{attribute 'linkalways'} 
{attribute 'no_explicit_call' := 'This FB is a CLASS and must be accessed using methods or properties'}
{attribute 'enable_dynamic_creation'}
FUNCTION_BLOCK Node_ContainerType_Vector_ITcVnImage EXTENDS Node
VAR
    out : _GUID;
END_VAR

METHOD PUBLIC  Clone : I_Node
VAR
	pNode : POINTER TO Node_ContainerType_Vector_ITcVnImage;
END_VAR
pNode := __NEW(Node_ContainerType_Vector_ITcVnImage);
Clone := pNode^;
END_METHOD

METHOD FB_init : BOOL
VAR_INPUT
	bInitRetains : BOOL; // if TRUE, the retain variables are initialized (warm start / cold start)
	bInCopyCode : BOOL;  // if TRUE, the instance afterwards gets moved into the copy code (online change)
END_VAR
AddOutput('out', out);
END_METHOD

METHOD PROTECTED OnExecute
out.Value := ContainerType_Vector_ITcVnImage;
END_METHOD

END_FUNCTION_BLOCK

(* stored: Version 1.1.0.1, ProductVersion 3.1.4026.17
   POU Node_ContainerType_Vector_ITcVnImage: Id {d99a62e1-c34a-0c88-0789-0f8a727a2aa7}, SpecialFunc None
   Folder Constructor: Id {77356306-f1ea-0116-04aa-6b0d3434c50a}
   Method Clone: Id {bc53d0b9-62fc-0f2c-3a7b-fe263fddab8f}
   Method FB_init: Id {c6402070-8556-0233-1ba3-b0bc6d5f63dd}
   Method OnExecute: Id {aacf9ed7-9f0f-05f7-1e41-7edf40c33269} *)
